// TIA Portal V19 export
TYPE "LUC_typeSignalStackConfiguration"
TITLE = LUC_typeSignalStackState
// Bahviour settings for the signal stack - machine modes
// stored: Access Published
   STRUCT
      undefined { ExternalWritable := 'False'} : "LUC_typeSignalStackStateBehaviour";   // Stack light configuration for state "Undefined"
      clearing { ExternalWritable := 'False'} : "LUC_typeSignalStackStateBehaviour";   // Stack light configuration for state "Clearing"
      stopped { ExternalWritable := 'False'} : "LUC_typeSignalStackStateBehaviour";   // Stack light configuration for state "Stopped"
      starting { ExternalWritable := 'False'} : "LUC_typeSignalStackStateBehaviour";   // Stack light configuration for state "Starting"
      idle { ExternalWritable := 'False'} : "LUC_typeSignalStackStateBehaviour";   // Stack light configuration for state "Idle"
      suspended { ExternalWritable := 'False'} : "LUC_typeSignalStackStateBehaviour";   // Stack light configuration for state "Suspended"
      execute { ExternalWritable := 'False'} : "LUC_typeSignalStackStateBehaviour";   // Stack light configuration for state "Execute"
      stopping { ExternalWritable := 'False'} : "LUC_typeSignalStackStateBehaviour";   // Stack light configuration for state "Stopping"
      aborting { ExternalWritable := 'False'} : "LUC_typeSignalStackStateBehaviour";   // Stack light configuration for state "Aborting"
      aborted { ExternalWritable := 'False'} : "LUC_typeSignalStackStateBehaviour";   // Stack light configuration for state "Aborted"
      holding { ExternalWritable := 'False'} : "LUC_typeSignalStackStateBehaviour";   // Stack light configuration for state "Holding"
      held { ExternalWritable := 'False'} : "LUC_typeSignalStackStateBehaviour";   // Stack light configuration for state "Held"
      unholding { ExternalWritable := 'False'} : "LUC_typeSignalStackStateBehaviour";   // Stack light configuration for state "Unholding"
      suspending { ExternalWritable := 'False'} : "LUC_typeSignalStackStateBehaviour";   // Stack light configuration for state "Suspending"
      unsuspending { ExternalWritable := 'False'} : "LUC_typeSignalStackStateBehaviour";   // Stack light configuration for state "Unsuspending"
      resetting { ExternalWritable := 'False'} : "LUC_typeSignalStackStateBehaviour";   // Stack light configuration for state "Resetting"
      completing { ExternalWritable := 'False'} : "LUC_typeSignalStackStateBehaviour";   // Stack light configuration for state "Completing"
      completed { ExternalWritable := 'False'} : "LUC_typeSignalStackStateBehaviour";   // Stack light configuration for state "Completed"
   END_STRUCT;
   // // undefined.static : Configuration of static lights for "undefined" state
   // // undefined.flashing : Configuration of flashing lights for "undefined" state
   // undefined.flashing.red := TRUE;
   // // clearing.static : Configuration of static lights for "clearing" state
   // // clearing.flashing : Configuration of flashing lights for "clearing" state
   // clearing.flashing.red := TRUE;
   // // stopped.static : Configuration of static lights for "stopped" state
   // stopped.static.red := TRUE;
   // // stopped.flashing : Configuration of flashing lights for "stopped" state
   // // starting.static : Configuration of static lights for "starting" state
   // starting.static.green := TRUE;
   // // starting.flashing : Configuration of flashing lights for "starting" state
   // // idle.static : Configuration of static lights for "idle" state
   // // idle.flashing : Configuration of flashing lights for "idle" state
   // idle.flashing.green := TRUE;
   // // suspended.static : Configuration of static lights for "suspended" state
   // suspended.static.yellow := TRUE;
   // // suspended.flashing : Configuration of flashing lights for "suspended" state
   // // execute.static : Configuration of static lights for "execute" state
   // execute.static.green := TRUE;
   // // execute.flashing : Configuration of flashing lights for "execute" state
   // // stopping.static : Configuration of static lights for "stopping" state
   // stopping.static.red := TRUE;
   // // stopping.flashing : Configuration of flashing lights for "stopping" state
   // // aborting.static : Configuration of static lights for "aborting" state
   // // aborting.flashing : Configuration of flashing lights for "aborting" state
   // aborting.flashing.red := TRUE;
   // // aborted.static : Configuration of static lights for "aborted" state
   // // aborted.flashing : Configuration of flashing lights for "aborted" state
   // aborted.flashing.red := TRUE;
   // // holding.static : Configuration of static lights for "holding" state
   // // holding.flashing : Configuration of flashing lights for "holding" state
   // holding.flashing.blue := TRUE;
   // // held.static : Configuration of static lights for "held" state
   // held.static.blue := TRUE;
   // // held.flashing : Configuration of flashing lights for "held" state
   // // unholding.static : Configuration of static lights for "unholding" state
   // unholding.static.green := TRUE;
   // // unholding.flashing : Configuration of flashing lights for "unholding" state
   // // suspending.static : Configuration of static lights for "suspending" state
   // // suspending.flashing : Configuration of flashing lights for "suspending" state
   // suspending.flashing.yellow := TRUE;
   // // unsuspending.static : Configuration of static lights for "unsuspending" state
   // unsuspending.static.green := TRUE;
   // // unsuspending.flashing : Configuration of flashing lights for "unsuspending" state
   // // resetting.static : Configuration of static lights for "resetting" state
   // resetting.static.red := TRUE;
   // // resetting.flashing : Configuration of flashing lights for "resetting" state
   // // completing.static : Configuration of static lights for "completing" state
   // completing.static.green := TRUE;
   // // completing.flashing : Configuration of flashing lights for "completing" state
   // // completed.static : Configuration of static lights for "completed" state
   // completed.static.red := TRUE;
   // // completed.flashing : Configuration of flashing lights for "completed" state
END_TYPE
